(* Logix 5000 project; controller CLASE_1 Emulate 5570 rev 28.11; software revision 28.02; part 4 of 15 *)
(* tags used below, declared in another part *)
   Inp_PV : BOOL;   // Input Signal (process variable) from Sensor
   Inp_PVBad : BOOL;   // Input Comm Status or Quality 1=Bad, 0=OK
   Inp_Target : BOOL;   // Target State of Input (Disagree Status if not in Target State)
   Inp_Sim : BOOL;   // 1=Use simulated PV (Set_SimPV); 0=Use Input (Inp_PV)
   Cfg_NoSubstPV : BOOL;   // 1=Disallow selection of Substitute PV
   Cfg_Debounce : REAL;   // Minimum time Input Sts must maintain state (sec)
   MSet_SubstPV : BOOL;   // Maintenance-Entered Substitute PV
   Set_SimPV : BOOL;   // PV used in Simulation (Inp_Sim=1)
   MCmd_SubstPV : BOOL;   // Maintenance Command to use Substitute PV (override input)
   MCmd_InpPV : BOOL;   // Maintenance Command to use Input PV (normal)
   OCmd_ResetAckAll : BOOL;   // Operator Command to Reset and Acknowledge all Alarms
   SrcQ_IO : SINT;   // Source and Quality of primary I/O (enumeration)
   SrcQ : SINT;   // Source and Quality of primary Val/Sts (enumeration)
   Val_Sts : SINT;   // Device Confirmed Sts 0=PV Good, 6=PV Bad, 7=Substitute PV
   Val_Fault : SINT;   // Device Fault Status 0=none, 16=Tgt Disagree, 34=CfgErr
   Val_Notify : SINT;   // Current Alarm Level and Acknowledgement (enumeration)
   Sts : BOOL;   // Discrete Input Status (incl. Debounce, Manual Override, if used)
   Sts_PV : BOOL;   // Discrete Input Status (actual, not subject to Override)
   Sts_SubstPV : BOOL;   // 1=Using Substitute PV (Input being overridden)
   Sts_InpPV : BOOL;   // 1=Using Input PV (normal)
   Sts_PVBad : BOOL;   // Input Comm Status/ Quality (0=OK, 1=Bad)
   Sts_MaintByp : BOOL;   // 1=Device has a Maintenance Bypass function active
   Sts_AlmInh : BOOL;   // 1=One or more Alarms Shelved, Disabled or Suppressed
   Err_Alarm : BOOL;   // 1=Error in Config: Alarm Min On Time, Shelf Time, Severity
   Sts_TgtDisagreeCmp : ALIAS FOR TgtDisagreeGate.Inp;   // Input vs. Target comparicon result 1=Disagree
   Sts_TgtDisagree : ALIAS FOR TgtDisagree.Inp;   // 1=Input is not in Target state
   Rdy_SubstPV : BOOL;   // 1=Ready for MCmd_SubstPV
   Rdy_InpPV : BOOL;   // 1=Ready for MCmd_InpPV
   Rdy_ResetAckAll : BOOL;   // 1=At least one Alarm requires Acknowledgement
   P_DIn : BOOL;   // Unique Parameter Name for auto - discovery
   TgtDisagree : P_Alarm;   // Target Disagree Alarm
   Wrk_FallT : TIMER;   // Timer to ensure Status LOW time on falling edge
   Wrk_RiseT : TIMER;   // Timer to ensure Status HIGH time on rising edge
   Wrk_SubstPV : BOOL;   // Internal flag: Using Substitute PV
   Cfg_1StText : STRING_8;   // Text to display in PV=1 State
   Cfg_0StText : STRING_8;   // Text to display in PV=0 State
   Wrk_Fault : SINT;   // Buffer for building Val_Fault
   Wrk_Status : SINT;   // Buffer for building Val_Sts
   Wrk_SrcQ : SINT;   // Register for building Source / Quality enumeration
   TgtDisagreeGate : P_Gate;   // Target Disagree Condition Gate/Delay
(* P_DIn, continued *)

ROUTINE Logic   (* ladder *)
// Normal Scan - status is updated and alarms are generated
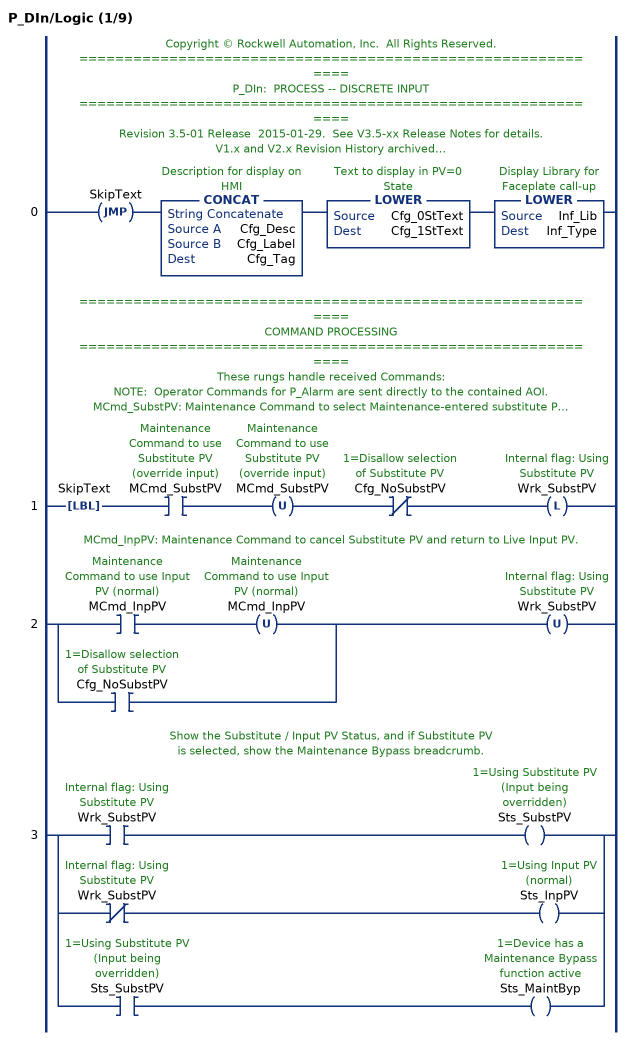
   // Copyright © Rockwell Automation, Inc.  All Rights Reserved.
   // ============================================================
   // P_DIn:  PROCESS -- DISCRETE INPUT
   // ============================================================
   // Revision 3.5-01 Release  2015-01-29.  See V3.5-xx Release Notes for details.
   // V1.x and V2.x Revision History archived.
   // V3.0-00  2013-06-30:  Added Inf_Lib. Uses P_Gate V3.0, P_Alarm V3.0.
   // V3.0-01  2013-07-30:  Modified Parameter descriptions only.
   // V3.0-02  2013-09-03:  Modified Parameter descriptions only.
   // V3.0-03  2013-10-30:  Corrected Parameter descriptions and default
   // configuration values for alarms only.
   // V3.1-00  2014-07-08:  Modified to use P_Alarm V3.1, add source/quality values (SrcQ).
   // V3.1-01  2014-09-03:  Unchanged, but using P_Alarm V3.1-01.
   // V3.1-02  2014-09-30:  Unchanged, but using P_Alarm V3.1-02.
   // V3.1-05  2016-01-22:  Unchanged, but using P_Gate V3.1-05.
   // V3.5-01  2016-01-29:  Unchanged, using P_Alarm, P_Gate V3.5-01.
   // ============================================================
   // This Instruction monitors a Discrete Input from a flow switch, motor overload,
   // or any other discrete signal, and provides:
   // *  Status, with configurable names for the 0- and 1-states
   // *  An Alarm "Gate" signal (with delay), used to enable an Alarm under appropriate process conditions
   // *  A "Target" input -- the Alarm is raised when the input is not in the same
   // state as the Target for a configurable period of time
   // * Input debounce for both the rising and falling transitions
   // * Commands to inhibit or enable alarms
   // * Monitoring of input communication status
   // * Setting of a simulated input signal for process simulation
   // * Selection of Substitute PV (by Maintenance personnel) or normal PV
   // Alarm is provided by a P_Alarm AOI instance.
   // Status gating provided by P_Gate AOI instances.
   // ============================================================
   // SHOW LOCAL STRINGS
   // ============================================================
   // The STRINGs containing the text associated with each instance of this
   // instruction cannot be Input or Output Parameters, because STRINGs are not
   //  'atomic' types. (Inputs and Outputs must be SINT, INT, DINT, REAL, or BOOL.)
   // In order to make it easier to find and configure these STRINGs, this rung
   // was added.  THE JMP (and the LBL on the following rung)
   // MUST NOT BE REMOVED!!!
   // To view the STRINGs, go to the instruction instance (in LD or FBD), RIGHT-click
   // to bring up the context menu and select "Open Instruction Logic".
   // This rung will appear with the STRING values for the selected instance.
   // You may double-click the STRING values here to modify them as well.
   // #####  V3.0-00  2013-06-30:  Added Inf_Lib.  #####
   0: JMP(SkipText)CONCAT(Cfg_Desc,Cfg_Label,Cfg_Tag)LOWER(Cfg_0StText,Cfg_1StText)LOWER(Inf_Lib,Inf_Type);
   // ============================================================
   // COMMAND PROCESSING
   // ============================================================
   // These rungs handle received Commands:
   // NOTE:  Operator Commands for P_Alarm are sent directly to the contained AOI.
   // MCmd_SubstPV: Maintenance Command to select Maintenance-entered substitute PV
   // Do not allow this Command if Cfg_NoSubstPV is set.
   1: LBL(SkipText)XIC(MCmd_SubstPV)OTU(MCmd_SubstPV)XIO(Cfg_NoSubstPV)OTL(Wrk_SubstPV);
   // MCmd_InpPV: Maintenance Command to cancel Substitute PV and return to Live Input PV.
   2: [XIC(MCmd_InpPV) OTU(MCmd_InpPV) ,XIC(Cfg_NoSubstPV) ]OTU(Wrk_SubstPV);
   // Show the Substitute / Input PV Status, and if Substitute PV
   // is selected, show the Maintenance Bypass breadcrumb.
   3: [XIC(Wrk_SubstPV) OTE(Sts_SubstPV) ,XIO(Wrk_SubstPV) OTE(Sts_InpPV) ,XIC(Sts_SubstPV) OTE(Sts_MaintByp) ];
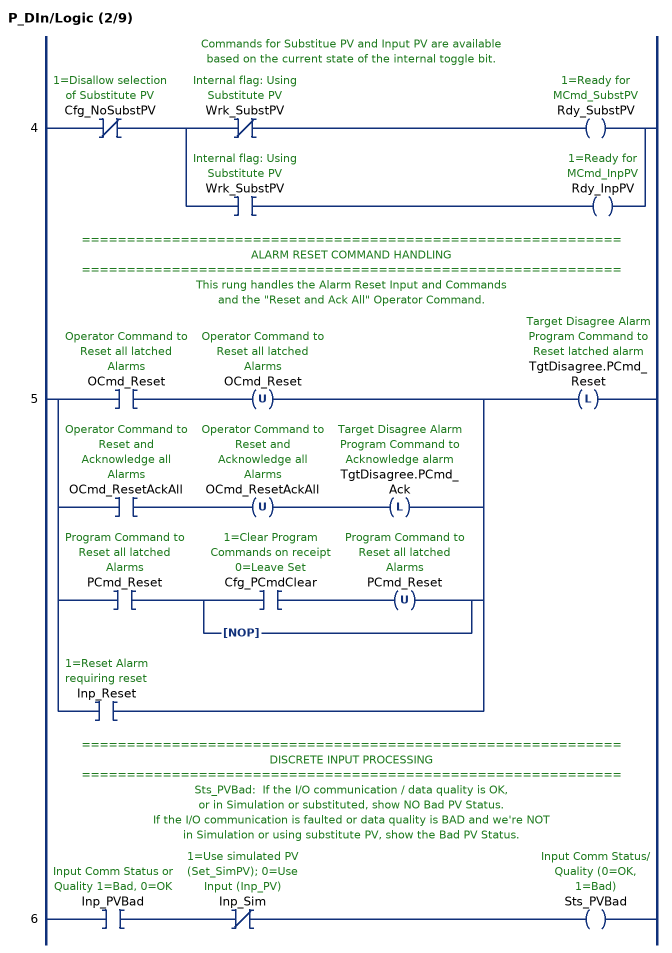
   // Commands for Substitue PV and Input PV are available
   // based on the current state of the internal toggle bit.
   4: XIO(Cfg_NoSubstPV)[XIO(Wrk_SubstPV) OTE(Rdy_SubstPV) ,XIC(Wrk_SubstPV) OTE(Rdy_InpPV) ];
   // ============================================================
   // ALARM RESET COMMAND HANDLING
   // ============================================================
   // This rung handles the Alarm Reset Input and Commands
   // and the "Reset and Ack All" Operator Command.
   5: [XIC(OCmd_Reset) OTU(OCmd_Reset) ,XIC(OCmd_ResetAckAll) OTU(OCmd_ResetAckAll) OTL(TgtDisagree.PCmd_Ack) ,XIC(PCmd_Reset) [XIC(Cfg_PCmdClear) OTU(PCmd_Reset) ,NOP() ] ,XIC(Inp_Reset) ]OTL(TgtDisagree.PCmd_Reset);
   // ============================================================
   // DISCRETE INPUT PROCESSING
   // ============================================================
   // Sts_PVBad:  If the I/O communication / data quality is OK,
   // or in Simulation or substituted, show NO Bad PV Status.
   // If the I/O communication is faulted or data quality is BAD and we're NOT
   // in Simulation or using substitute PV, show the Bad PV Status.
   6: XIC(Inp_PVBad)XIO(Inp_Sim)OTE(Sts_PVBad);
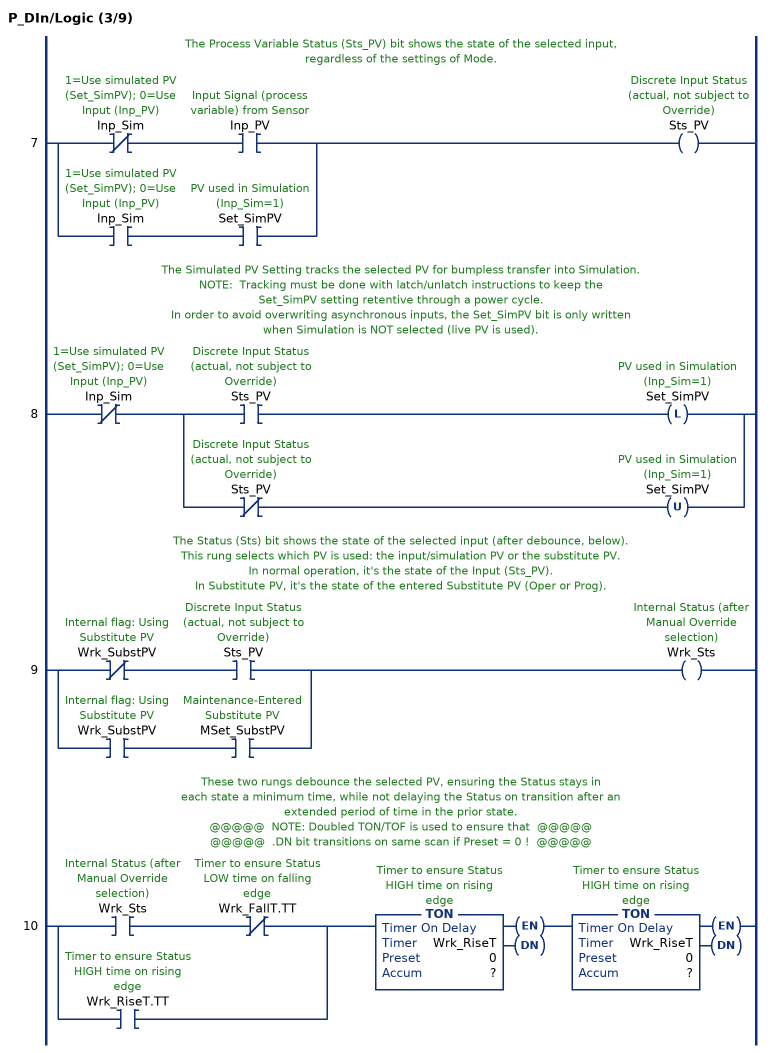
   // The Process Variable Status (Sts_PV) bit shows the state of the selected input,
   // regardless of the settings of Mode.
   7: [XIO(Inp_Sim) XIC(Inp_PV) ,XIC(Inp_Sim) XIC(Set_SimPV) ]OTE(Sts_PV);
   // The Simulated PV Setting tracks the selected PV for bumpless transfer into Simulation.
   // NOTE:  Tracking must be done with latch/unlatch instructions to keep the
   // Set_SimPV setting retentive through a power cycle.
   // In order to avoid overwriting asynchronous inputs, the Set_SimPV bit is only written
   // when Simulation is NOT selected (live PV is used).
   8: XIO(Inp_Sim)[XIC(Sts_PV) OTL(Set_SimPV) ,XIO(Sts_PV) OTU(Set_SimPV) ];
   // The Status (Sts) bit shows the state of the selected input (after debounce, below).
   // This rung selects which PV is used: the input/simulation PV or the substitute PV.
   // In normal operation, it's the state of the Input (Sts_PV).
   // In Substitute PV, it's the state of the entered Substitute PV (Oper or Prog).
   9: [XIO(Wrk_SubstPV) XIC(Sts_PV) ,XIC(Wrk_SubstPV) XIC(MSet_SubstPV) ]OTE(Wrk_Sts);
   // These two rungs debounce the selected PV, ensuring the Status stays in
   // each state a minimum time, while not delaying the Status on transition after an
   // extended period of time in the prior state.
   // @@@@@  NOTE: Doubled TON/TOF is used to ensure that  @@@@@
   // @@@@@  .DN bit transitions on same scan if Preset = 0 !  @@@@@
   10: [XIC(Wrk_Sts) XIO(Wrk_FallT.TT) ,XIC(Wrk_RiseT.TT) ]TON(Wrk_RiseT,?,?)TON(Wrk_RiseT,?,?);
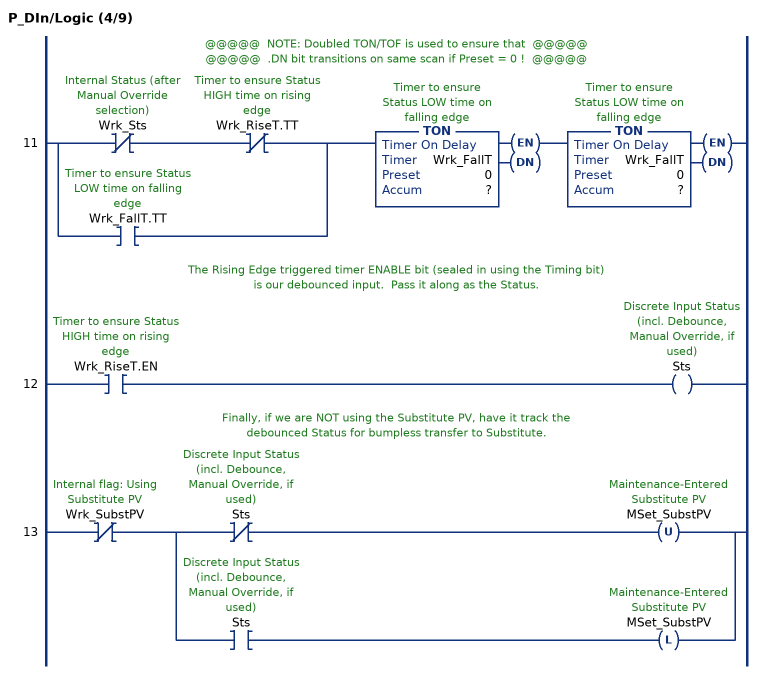
   // @@@@@  NOTE: Doubled TON/TOF is used to ensure that  @@@@@
   // @@@@@  .DN bit transitions on same scan if Preset = 0 !  @@@@@
   11: [XIO(Wrk_Sts) XIO(Wrk_RiseT.TT) ,XIC(Wrk_FallT.TT) ]TON(Wrk_FallT,?,?)TON(Wrk_FallT,?,?);
   // The Rising Edge triggered timer ENABLE bit (sealed in using the Timing bit)
   // is our debounced input.  Pass it along as the Status.
   12: XIC(Wrk_RiseT.EN)OTE(Sts);
   // Finally, if we are NOT using the Substitute PV, have it track the
   // debounced Status for bumpless transfer to Substitute.
   13: XIO(Wrk_SubstPV)[XIO(Sts) OTU(MSet_SubstPV) ,XIC(Sts) OTL(MSet_SubstPV) ];
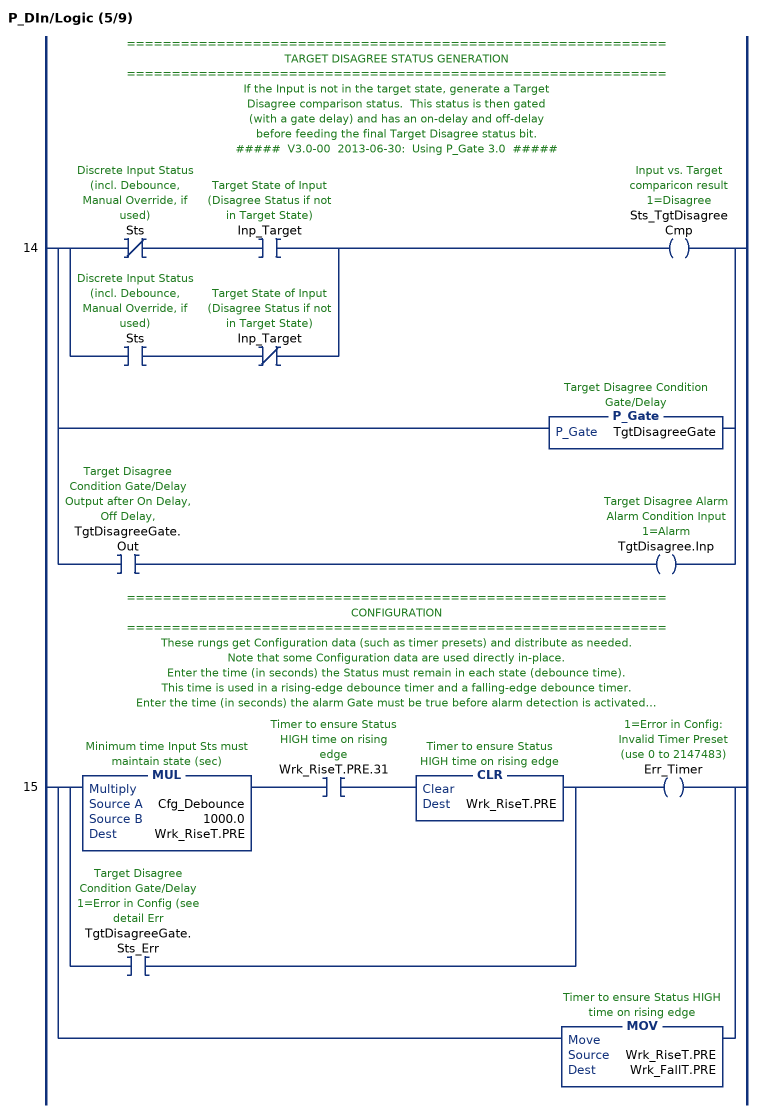
   // ============================================================
   // TARGET DISAGREE STATUS GENERATION
   // ============================================================
   // If the Input is not in the target state, generate a Target
   // Disagree comparison status.  This status is then gated
   // (with a gate delay) and has an on-delay and off-delay
   // before feeding the final Target Disagree status bit.
   // #####  V3.0-00  2013-06-30:  Using P_Gate 3.0  #####
   14: [[XIO(Sts) XIC(Inp_Target) ,XIC(Sts) XIO(Inp_Target) ] OTE(Sts_TgtDisagreeCmp) ,P_Gate(TgtDisagreeGate) ,XIC(TgtDisagreeGate.Out) OTE(TgtDisagree.Inp) ];
   // ============================================================
   // CONFIGURATION
   // ============================================================
   // These rungs get Configuration data (such as timer presets) and distribute as needed.
   // Note that some Configuration data are used directly in-place.
   // Enter the time (in seconds) the Status must remain in each state (debounce time).
   // This time is used in a rising-edge debounce timer and a falling-edge debounce timer.
   // Enter the time (in seconds) the alarm Gate must be true before alarm detection is activated.
   // Enter the On-Delay and Off-Delay times (in seconds) for the Target Disagree Status
   // (which feeds the Target Disagree Alarm).
   // If the timer preset calcuated wraps negative (more than 2.14... million seconds), then establish
   // a valid limit value for the Preset.  Note that a negative timer preset will fault the controller!!!
   // #####  V3.0-00  2013-06-30:  Using P_Gate 3.0  #####
   15: [[MUL(Cfg_Debounce,1000.0,Wrk_RiseT.PRE) XIC(Wrk_RiseT.PRE.31) CLR(Wrk_RiseT.PRE) ,XIC(TgtDisagreeGate.Sts_Err) ] OTE(Err_Timer) ,MOV(Wrk_RiseT.PRE,Wrk_FallT.PRE) ];
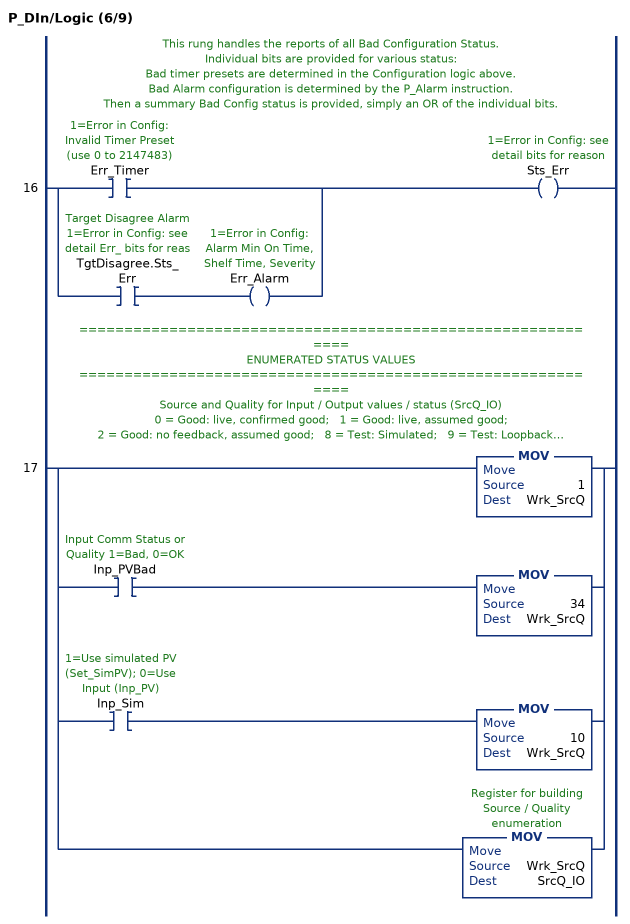
   // This rung handles the reports of all Bad Configuration Status.
   // Individual bits are provided for various status:
   // Bad timer presets are determined in the Configuration logic above.
   // Bad Alarm configuration is determined by the P_Alarm instruction.
   // Then a summary Bad Config status is provided, simply an OR of the individual bits.
   16: [XIC(Err_Timer) ,XIC(TgtDisagree.Sts_Err) OTE(Err_Alarm) ]OTE(Sts_Err);
   // ============================================================
   // ENUMERATED STATUS VALUES
   // ============================================================
   // Source and Quality for Input / Output values / status (SrcQ_IO)
   // 0 = Good: live, confirmed good;   1 = Good: live, assumed good;
   // 2 = Good: no feedback, assumed good;   8 = Test: Simulated;   9 = Test: Loopback;
   // 10 = Test: Manually Entered;   16 = Uncertain: Live, off-spec;
   // 17 = Uncertain, Substituted at Device / Bus;   18 = Uncertain, Substituted at AOI;
   // 19 = Uncertain, using last known good;    20 = Uncertain, using replacement value;
   // 32 = Bad, Signal Failure;   33 = Bad, Channel Fault;
   // 34 = Bad, Module / Comms Fault;   35 = Bad, Invalid Configuration
   // #####  V3.1-00  2014-06-30:  Added rung for Source/Quality enumerations.  #####
   17: [MOV(1,Wrk_SrcQ) ,XIC(Inp_PVBad) MOV(34,Wrk_SrcQ) ,XIC(Inp_Sim) MOV(10,Wrk_SrcQ) ,MOV(Wrk_SrcQ,SrcQ_IO) ];
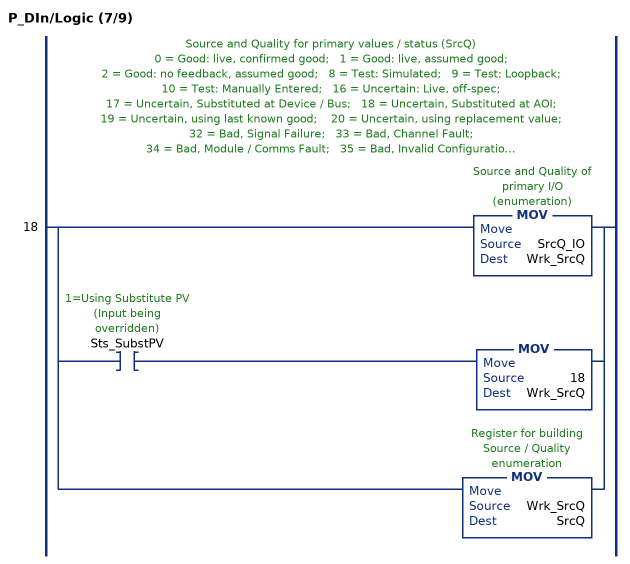
   // Source and Quality for primary values / status (SrcQ)
   // 0 = Good: live, confirmed good;   1 = Good: live, assumed good;
   // 2 = Good: no feedback, assumed good;   8 = Test: Simulated;   9 = Test: Loopback;
   // 10 = Test: Manually Entered;   16 = Uncertain: Live, off-spec;
   // 17 = Uncertain, Substituted at Device / Bus;   18 = Uncertain, Substituted at AOI;
   // 19 = Uncertain, using last known good;    20 = Uncertain, using replacement value;
   // 32 = Bad, Signal Failure;   33 = Bad, Channel Fault;
   // 34 = Bad, Module / Comms Fault;   35 = Bad, Invalid Configuration
   // #####  V3.1-00  2014-06-30:  Added rung for Source/Quality enumerations.  #####
   18: [MOV(SrcQ_IO,Wrk_SrcQ) ,XIC(Sts_SubstPV) MOV(18,Wrk_SrcQ) ,MOV(Wrk_SrcQ,SrcQ) ];
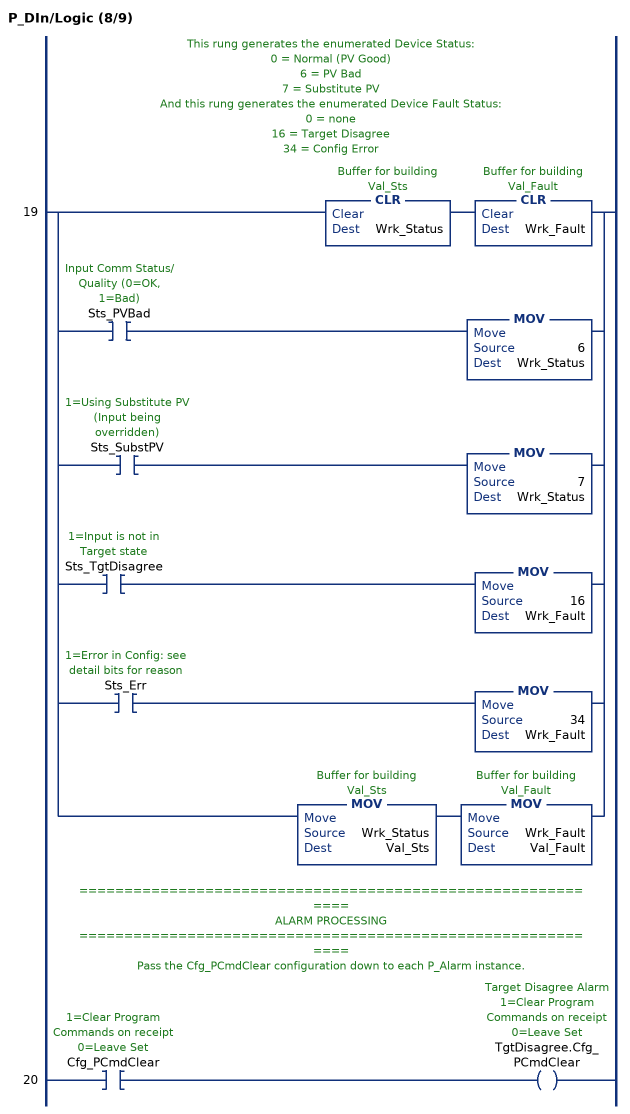
   // This rung generates the enumerated Device Status:
   // 0 = Normal (PV Good)
   // 6 = PV Bad
   // 7 = Substitute PV
   // And this rung generates the enumerated Device Fault Status:
   // 0 = none
   // 16 = Target Disagree
   // 34 = Config Error
   19: [CLR(Wrk_Status) CLR(Wrk_Fault) ,XIC(Sts_PVBad) MOV(6,Wrk_Status) ,XIC(Sts_SubstPV) MOV(7,Wrk_Status) ,XIC(Sts_TgtDisagree) MOV(16,Wrk_Fault) ,XIC(Sts_Err) MOV(34,Wrk_Fault) ,MOV(Wrk_Status,Val_Sts) MOV(Wrk_Fault,Val_Fault) ];
   // ============================================================
   // ALARM PROCESSING
   // ============================================================
   // Pass the Cfg_PCmdClear configuration down to each P_Alarm instance.
   20: XIC(Cfg_PCmdClear)OTE(TgtDisagree.Cfg_PCmdClear);
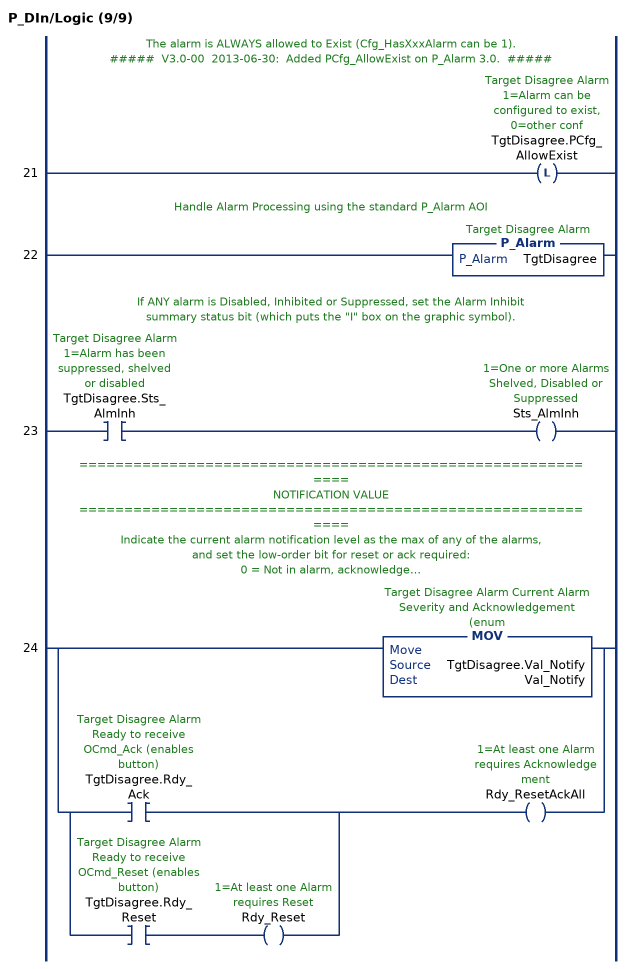
   // The alarm is ALWAYS allowed to Exist (Cfg_HasXxxAlarm can be 1).
   // #####  V3.0-00  2013-06-30:  Added PCfg_AllowExist on P_Alarm 3.0.  #####
   21: OTL(TgtDisagree.PCfg_AllowExist);
   // Handle Alarm Processing using the standard P_Alarm AOI
   22: P_Alarm(TgtDisagree);
   // If ANY alarm is Disabled, Inhibited or Suppressed, set the Alarm Inhibit
   // summary status bit (which puts the "I" box on the graphic symbol).
   23: XIC(TgtDisagree.Sts_AlmInh)OTE(Sts_AlmInh);
   // ============================================================
   // NOTIFICATION VALUE
   // ============================================================
   // Indicate the current alarm notification level as the max of any of the alarms,
   // and set the low-order bit for reset or ack required:
   // 0 = Not in alarm, acknowledged
   // 1 = Not in alarm, unacknowledged or reset required
   // 2 = Low severity alarm, acknowledged
   // 3 = Low severity alarm, unacknowledged
   // 4 = Medium severity alarm, acknowledged
   // 5 = Medium severity alarm, unacknowledged
   // 6 = High severity alarm, acknowledged
   // 7 = High severity alarm, unacknowledged
   // 8 = Urgent severity alarm, acknowledged
   // 9 = Urgent severity alarm, unacknowledged
   // #####  V3.1-00  2014-06-30:  Separated Reset Reqd functions from Val_Notify  #####
   24: [MOV(TgtDisagree.Val_Notify,Val_Notify) ,[XIC(TgtDisagree.Rdy_Ack) ,XIC(TgtDisagree.Rdy_Reset) OTE(Rdy_Reset) ] OTE(Rdy_ResetAckAll) ];
END_ROUTINE

ROUTINE Prescan   (* ladder *)
// Clear "lurking" Commands
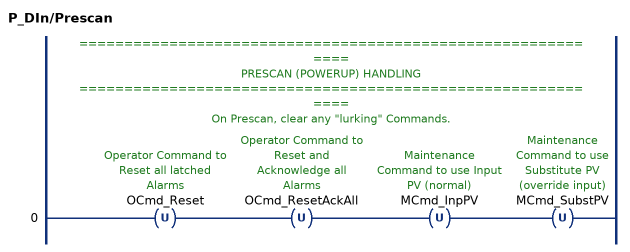
   // ============================================================
   // PRESCAN (POWERUP) HANDLING
   // ============================================================
   // On Prescan, clear any "lurking" Commands.
   0: OTU(OCmd_Reset)OTU(OCmd_ResetAckAll)OTU(MCmd_InpPV)OTU(MCmd_SubstPV);
END_ROUTINE
END_ADD_ON_INSTRUCTION

ADD_ON_INSTRUCTION P_FT_Primer_Orden_AOI   (* revision 1.0 *)
// Simula el comportamiento de una Función de Transferencia de primer orden.
// G(s) = Kp/(Tao*s + 1)
VAR_INPUT
   Kp : REAL; {visible}   // Ganancia proporcional de la FT.
   Tao : REAL; {visible}   // Tao de la FT (en segundos).
   Inp_Sistema : REAL; {visible}   // Entrada de la FT.
END_VAR
VAR_OUTPUT
   Out_Sistema : REAL; {visible}   // Salida de la FT.
END_VAR
VAR_INPUT
   Tiempo_muerto : REAL; {visible}   // Tiempo muerto (en segundos).
   Inp_Disturbio : REAL; {visible}   // Permite simular un disturbio en el sistema.
   FT_EnableIN : BOOL := 1; {visible}   // Bit para ejecutar algoritmo de la FT.
   FT_Bias : REAL; {visible}   // Simula condición de proceso. (In*Gain) + Bias.
END_VAR
VAR
   DEDT_01 : DEADTIME := (Gain := 1.0, RTSTime := 1); {access None}
   LDLG_01 : LEAD_LAG := (Gain := 1.0, RTSTime := 1); {access None}
   FT : LEAD_LAG := (Gain := 1.0, RTSTime := 1);   // Simula FT de Primer Orden.
   Tm : DEADTIME := (Gain := 1.0, RTSTime := 1); {access None}   // Simula Tiempo muerto.
   Tm_muestreo : REAL[1000]; {access None}   // Array para guardar valores previos al Tiempo muestro.
   ADD_01 : FBD_MATH; {access None}
   __l01D9873C3019917B : REAL; {access None}
   __l01D9933530198D26 : BOOL; {access None}
   __l01D9DEFB3019BCF5 : REAL; {access None}
   __l01D9CACD3019D0A3 : REAL; {access None}
   __l01D9EFCA30199939 : REAL; {access None}
   __l01D9E71B3019C2AC : REAL; {access None}
   __l01D9EBF23019A41E : REAL; {access None}
END_VAR

ROUTINE Logic   (* function block diagram *)
   SHEET 1
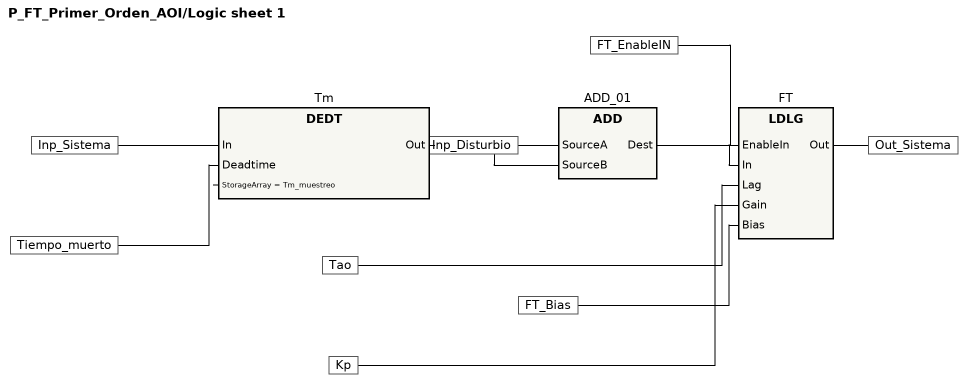
   Tm : DEDT(In := Inp_Sistema, Deadtime := Tiempo_muerto, StorageArray := Tm_muestreo);
   ADD_01 : ADD(SourceA := Inp_Disturbio, SourceB := Tm.Out);
   FT : LDLG(EnableIn := FT_EnableIN, In := ADD_01.Dest, Lag := Tao, Gain := Kp, Bias := FT_Bias);
   Out_Sistema := FT.Out;
END_ROUTINE
END_ADD_ON_INSTRUCTION

ADD_ON_INSTRUCTION P_Gate   (* revision 3.5 01 Release, vendor Rockwell Automation, ExecutePrescan, ExecuteEnableInFalse *)
// Condition Gate/Delay
// Revision note:
// See V3.5-xx Release Notes for details. Unchanged, up-rev only for V3.5 Library.
// Help:
// Copyright © Rockwell Automation, Inc.  All Rights Reserved.
// This Instruction provides a "gate" for a discrete Input signal and
// provides on-delay and off-delay timing for the gated signal.
// When the Gate input is true, the instruction Input is passed through
// to the Output, with on-delay and off-delay timing applied.
// When the Gate input is false, the Output is kept off
// (note: off-delay still applies!)
// This instruction is usually used between a comparison
// (analog threshold with deadband or discrete logic)
// and a P_Alarm instance, but may be used as a
// gated on-delay/off-delay timer generally.
// When EnableIn  is FALSE (e.g., on a false LD rung),
// the Input "Inp" is inverted.  Note that the Gate
// input (Inp_Gate) is NOT inverted!!!
VAR_INPUT
   Inp : BOOL; {visible}   // Input Condition: e.g., result of comparison
   Inp_Gate : BOOL := 1; {visible}   // Gate Input: 1=enable On Delay / Off Delay after Gate Delay, 0=disable
   Cfg_GateDly : DINT;   // Gate Delay (s): time after Gate Input true to enable On/Off Delay
   Cfg_OnDly : DINT;   // On Delay (s): If Gate Delay done, time Inp must be true to set Out true
   Cfg_OffDly : DINT;   // Off Delay (s): Time after Inp or Gate goes to 0 for Out to go to 0
END_VAR
VAR_OUTPUT
   Out : BOOL; {access Read Only, visible}   // Output after On Delay, Off Delay, enabled by Gate
   Sts_Gate : BOOL; {access Read Only, visible}   // 1=Gate Delay done, Output is enabled
   Sts_Err : BOOL; {access Read Only, visible}   // 1=Error in Config (see detail Err_ bits for reason), display icon
   Err_Timer : BOOL; {access Read Only}   // 1=Error in Config: On Delay, Off Delay, Gate Delay Time Invalid (use 0 to 2147483 s)
   P_Gate : BOOL;   // Unique Parameter Name for auto - discovery
END_VAR
VAR
   Wrk_OffDlyT : TIMER; {access Read Only}   // Off Delay Timer
   Wrk_OnDlyT : TIMER; {access Read Only}   // On Delay Timer
   Wrk_GateT : TIMER; {access Read Only}   // Gate Delay Timer
   Cfg_InpCond : STRING_20 := 'Input Condition';   // Displayed text of P_Gate's Input (Inp) Condition
   Inf_Lib : STRING_12 := 'RA-BAS'; {access Read Only}   // Display Library for Faceplate call-up
   Inf_Type : STRING_16 := 'P_Gate'; {access Read Only}   // Must contain AOI name, used for HMI and Information S/W
   Cfg_GateCond : STRING_20 := 'Gating Condition';   // Displayed text of P_Gate's Gating (Inp_Gate) Condition
   Inf_Tab : SINT;   // Tab to display (FTView ME)
END_VAR

ROUTINE EnableInFalse   (* ladder *)
// Same as main Logic routine, except Inp is inverted (for use in LD logic)  (Inp_Gate is NOT inverted!!!)
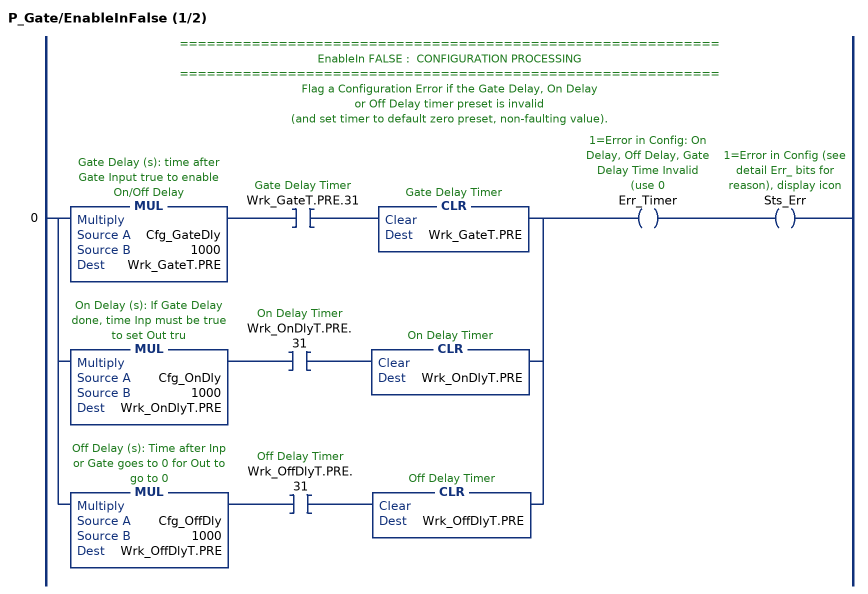
   // ============================================================
   // EnableIn FALSE :  CONFIGURATION PROCESSING
   // ============================================================
   // Flag a Configuration Error if the Gate Delay, On Delay
   // or Off Delay timer preset is invalid
   // (and set timer to default zero preset, non-faulting value).
   0: [MUL(Cfg_GateDly,1000,Wrk_GateT.PRE) XIC(Wrk_GateT.PRE.31) CLR(Wrk_GateT.PRE) ,MUL(Cfg_OnDly,1000,Wrk_OnDlyT.PRE) XIC(Wrk_OnDlyT.PRE.31) CLR(Wrk_OnDlyT.PRE) ,MUL(Cfg_OffDly,1000,Wrk_OffDlyT.PRE) XIC(Wrk_OffDlyT.PRE.31) CLR(Wrk_OffDlyT.PRE) ]OTE(Err_Timer)OTE(Sts_Err);
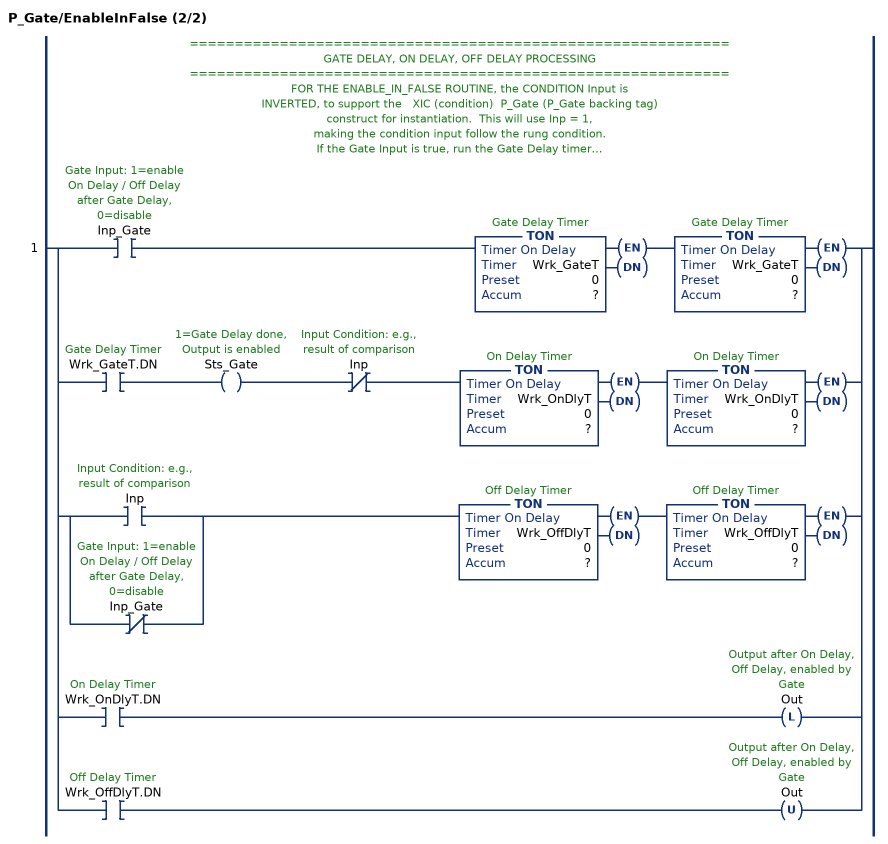
   // ============================================================
   // GATE DELAY, ON DELAY, OFF DELAY PROCESSING
   // ============================================================
   // FOR THE ENABLE_IN_FALSE ROUTINE, the CONDITION Input is
   // INVERTED, to support the   XIC (condition)  P_Gate (P_Gate backing tag)
   // construct for instantiation.  This will use Inp = 1,
   // making the condition input follow the rung condition.
   // If the Gate Input is true, run the Gate Delay timer.
   // Once the Gate Delay is complete, enable the
   // On Delay and Off Delay that follow the INVERTED input.
   // Report the Gate Delay status and the final Output status (after all delays).
   // @@@@@  NOTE: Doubled TONs are used to ensure that  @@@@@
   // @@@@@  .DN bit transitions on same scan if Preset = 0 !  @@@@@
   1: [XIC(Inp_Gate) TON(Wrk_GateT,?,?) TON(Wrk_GateT,?,?) ,XIC(Wrk_GateT.DN) OTE(Sts_Gate) XIO(Inp) TON(Wrk_OnDlyT,?,?) TON(Wrk_OnDlyT,?,?) ,[XIC(Inp) ,XIO(Inp_Gate) ] TON(Wrk_OffDlyT,?,?) TON(Wrk_OffDlyT,?,?) ,XIC(Wrk_OnDlyT.DN) OTL(Out) ,XIC(Wrk_OffDlyT.DN) OTU(Out) ];
END_ROUTINE

ROUTINE Logic   (* ladder *)
// Gate the input and apply on-delay and off-delay timing
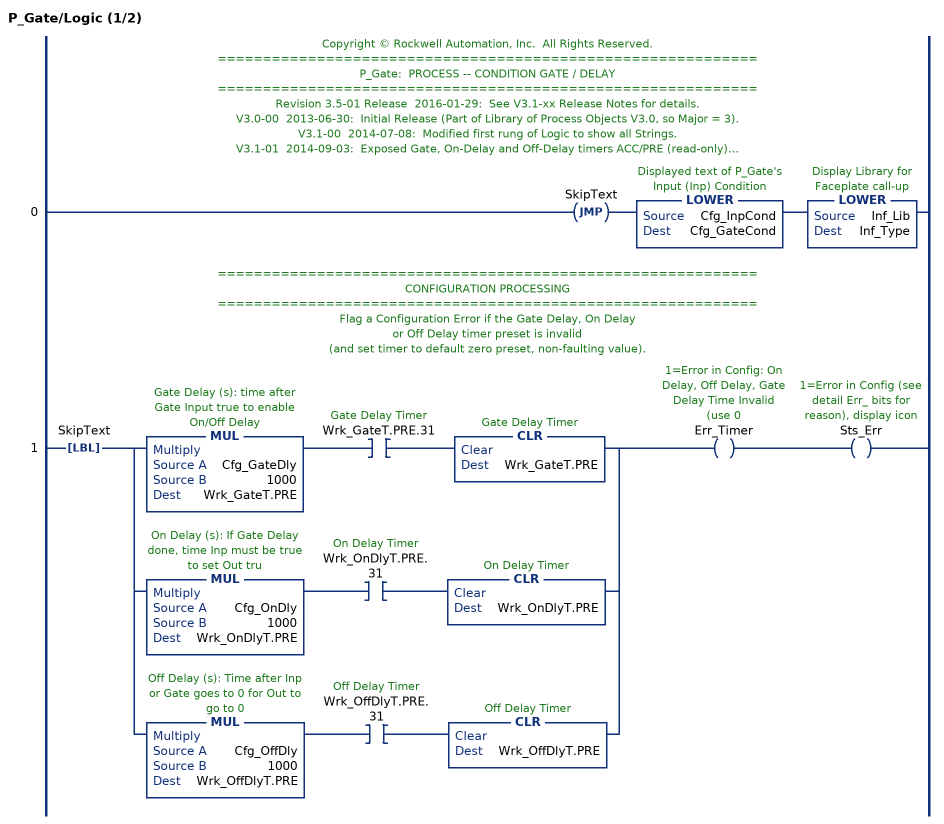
   // Copyright © Rockwell Automation, Inc.  All Rights Reserved.
   // ============================================================
   // P_Gate:  PROCESS -- CONDITION GATE / DELAY
   // ============================================================
   // Revision 3.5-01 Release  2016-01-29:  See V3.1-xx Release Notes for details.
   // V3.0-00  2013-06-30:  Initial Release (Part of Library of Process Objects V3.0, so Major = 3).
   // V3.1-00  2014-07-08:  Modified first rung of Logic to show all Strings.
   // V3.1-01  2014-09-03:  Exposed Gate, On-Delay and Off-Delay timers ACC/PRE (read-only).
   // V3.1-05  2016-01-22:  Corrected logic when using analog threshold with deadband.
   // V3.5-01  2016-01-29:  Unchanged, up-rev only for V3.5 Library.
   // ============================================================
   // This Instruction provides a "gate" for a discrete Input signal and
   // provides on-delay and off-delay timing for the gated signal.
   // When the Gate input is true, the instruction Input is passed through
   // to the Output, with on-delay and off-delay timing applied.
   // When the Gate input is false, the Output is kept off
   // (note: off-delay still applies!)
   // This instruction is usually used between a comparison
   // (analog threshold with deadband or discrete logic)
   // and a P_Alarm instance, but may be used as a
   // gated on-delay/off-delay timer generally.
   // When EnableIn  is FALSE (e.g., on a false LD rung),
   // the Input "Inp" is inverted.  Note that the Gate
   // input (Inp_Gate) is NOT inverted!!!
   // ============================================================
   // SHOW LOCAL STRINGS
   // ============================================================
   // The STRINGs containing the text associated with each instance of this
   // instruction cannot be Input or Output Parameters, because STRINGs are not
   //  'atomic' types. (Inputs and Outputs must be SINT, INT, DINT, REAL, or BOOL.)
   // In order to make it easier to find and configure these STRINGs, this rung
   // was added.  THE JMP (and the LBL on the following rung)
   // MUST NOT BE REMOVED!!!
   // To view the STRINGs, go to the instruction instance (in LD or FBD), RIGHT-click
   // to bring up the context menu and select "Open Instruction Logic".
   // This rung will appear with the STRING values for the selected instance.
   // You may double-click the STRING values here to modify them as well.
   // #####  V3.1-00  2014-07-08: Added Inf_Type to displayed Strings  #####
   0: JMP(SkipText)LOWER(Cfg_InpCond,Cfg_GateCond)LOWER(Inf_Lib,Inf_Type);
   // ============================================================
   // CONFIGURATION PROCESSING
   // ============================================================
   // Flag a Configuration Error if the Gate Delay, On Delay
   // or Off Delay timer preset is invalid
   // (and set timer to default zero preset, non-faulting value).
   1: LBL(SkipText)[MUL(Cfg_GateDly,1000,Wrk_GateT.PRE) XIC(Wrk_GateT.PRE.31) CLR(Wrk_GateT.PRE) ,MUL(Cfg_OnDly,1000,Wrk_OnDlyT.PRE) XIC(Wrk_OnDlyT.PRE.31) CLR(Wrk_OnDlyT.PRE) ,MUL(Cfg_OffDly,1000,Wrk_OffDlyT.PRE) XIC(Wrk_OffDlyT.PRE.31) CLR(Wrk_OffDlyT.PRE) ]OTE(Err_Timer)OTE(Sts_Err);
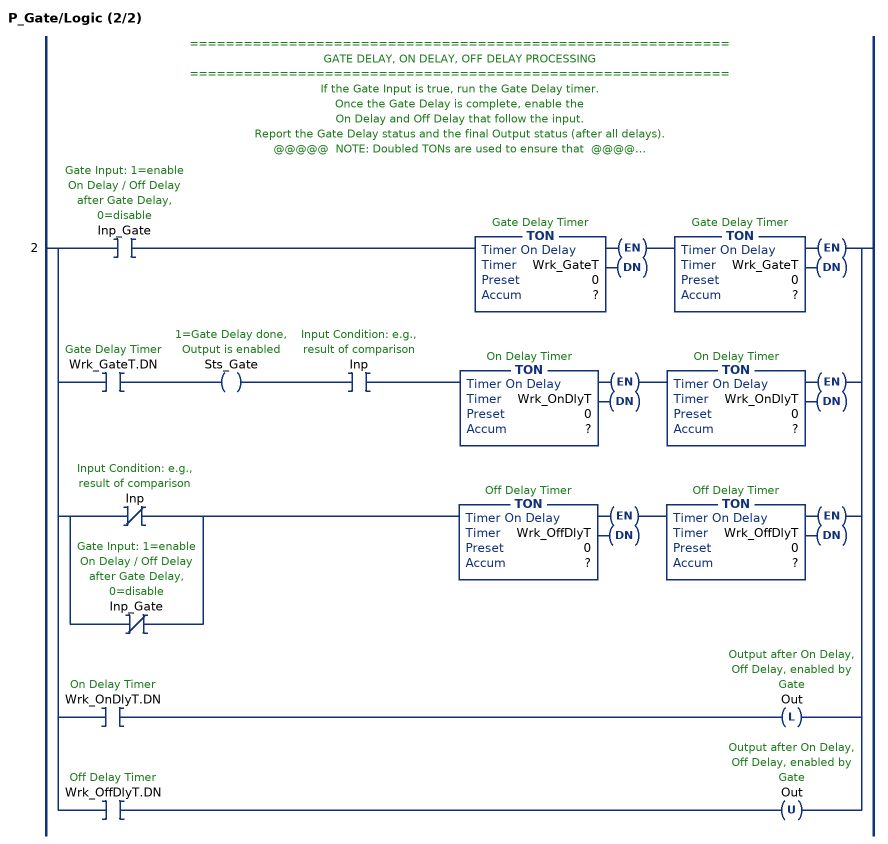
   // ============================================================
   // GATE DELAY, ON DELAY, OFF DELAY PROCESSING
   // ============================================================
   // If the Gate Input is true, run the Gate Delay timer.
   // Once the Gate Delay is complete, enable the
   // On Delay and Off Delay that follow the input.
   // Report the Gate Delay status and the final Output status (after all delays).
   // @@@@@  NOTE: Doubled TONs are used to ensure that  @@@@@
   // @@@@@  .DN bit transitions on same scan if Preset = 0 !  @@@@@
   2: [XIC(Inp_Gate) TON(Wrk_GateT,?,?) TON(Wrk_GateT,?,?) ,XIC(Wrk_GateT.DN) OTE(Sts_Gate) XIC(Inp) TON(Wrk_OnDlyT,?,?) TON(Wrk_OnDlyT,?,?) ,[XIO(Inp) ,XIO(Inp_Gate) ] TON(Wrk_OffDlyT,?,?) TON(Wrk_OffDlyT,?,?) ,XIC(Wrk_OnDlyT.DN) OTL(Out) ,XIC(Wrk_OffDlyT.DN) OTU(Out) ];
END_ROUTINE

ROUTINE Prescan   (* ladder *)
// Set the Gate Input to 1 (default value) on prescan
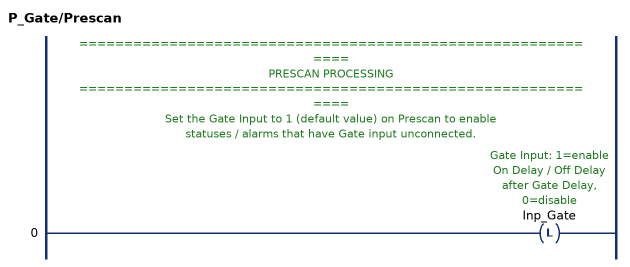
   // ============================================================
   // PRESCAN PROCESSING
   // ============================================================
   // Set the Gate Input to 1 (default value) on Prescan to enable
   // statuses / alarms that have Gate input unconnected.
   0: OTL(Inp_Gate);
END_ROUTINE
END_ADD_ON_INSTRUCTION

ADD_ON_INSTRUCTION P_Intlk   (* revision 3.5 05 Release, vendor Rockwell Automation, ExecutePrescan, ExecuteEnableInFalse *)
// Interlocks
// Revision note:
// See V3.5-xx Release Notes for details. Changed Nav Tags to user-defined STRING_NavTag type. Modified to maintain First Out indication until next stop.
// Help:
// Copyright © Rockwell Automation, Inc.  All Rights Reserved.
// This Instruction monitors up to 16 Interlock conditions.  It provides these features:
// *  The "OK" state of each Interlock Input is configurable.  By default,
//     each Input is 1 to trip, 0 when OK to run.
// *  Interlocks may be configured as Latched.  Latched Interlocks
//     require a Reset Command to clear.  The latching function can be
//     inhibited via a Latch Defeat input, for example, to avoid latching
//     Interlocks for a stopped motor.
// *  Interlocks may be configured as Bypassable; Non-Bypassable
//     Interlocks are reported separately so the destination object can
//     decide whether to bypass (ignore) bypassable interlocks, such
//     as in Maintenance Mode.
// *  First-Out reporting indicates the first condition that caused the
//     running equipment to be tripped.
// *  For each Interlock condition, a Tag may be defined for navigation.
//     Clicking the Interlock description will call up the associated Tag's
//     Faceplate.
VAR_INPUT
   Inp_Intlk00 : ALIAS FOR Wrk_Inp.0; {visible}   // Interlock Cond. 00, Stop if not in configured OK state
   Inp_Intlk01 : ALIAS FOR Wrk_Inp.1; {visible}   // Interlock Cond. 01, Stop if not in configured OK state
   Inp_Intlk02 : ALIAS FOR Wrk_Inp.2; {visible}   // Interlock Cond. 02, Stop if not in configured OK state
   Inp_Intlk03 : ALIAS FOR Wrk_Inp.3; {visible}   // Interlock Cond. 03, Stop if not in configured OK state
   Inp_Intlk04 : ALIAS FOR Wrk_Inp.4; {visible}   // Interlock Cond. 04, Stop if not in configured OK state
   Inp_Intlk05 : ALIAS FOR Wrk_Inp.5; {visible}   // Interlock Cond. 05, Stop if not in configured OK state
   Inp_Intlk06 : ALIAS FOR Wrk_Inp.6; {visible}   // Interlock Cond. 06, Stop if not in configured OK state
   Inp_Intlk07 : ALIAS FOR Wrk_Inp.7; {visible}   // Interlock Cond. 07, Stop if not in configured OK state
   Inp_Intlk08 : ALIAS FOR Wrk_Inp.8;   // Interlock Cond. 08, Stop if not in configured OK state
   Inp_Intlk09 : ALIAS FOR Wrk_Inp.9;   // Interlock Cond. 09, Stop if not in configured OK state
   Inp_Intlk10 : ALIAS FOR Wrk_Inp.10;   // Interlock Cond. 10, Stop if not in configured OK state
   Inp_Intlk11 : ALIAS FOR Wrk_Inp.11;   // Interlock Cond. 11, Stop if not in configured OK state
   Inp_Intlk12 : ALIAS FOR Wrk_Inp.12;   // Interlock Cond. 12, Stop if not in configured OK state
   Inp_Intlk13 : ALIAS FOR Wrk_Inp.13;   // Interlock Cond. 13, Stop if not in configured OK state
   Inp_Intlk14 : ALIAS FOR Wrk_Inp.14;   // Interlock Cond. 14, Stop if not in configured OK state
   Inp_Intlk15 : ALIAS FOR Wrk_Inp.15;   // Interlock Cond. 15, Stop if not in configured OK state
   Inp_BypActive : BOOL; {visible}   // 1=Interlock Bypassing is currently active
   Inp_LatchDefeat : BOOL; {visible}   // Latch Defeat 1=Do not latch inputs even if configured for latching
   Inp_Reset : BOOL; {visible}   // 1=Reset Latched Interlocks and First-Out
   Cfg_OKState : INT;   // Bits indicate which state (0 or 1) of each input is OK to run
   Cfg_Latched : INT;   // Set bits indicate which conditions are latched (sealed in)
   Cfg_Bypassable : INT;   // Set bits indicate which conditions can be bypassed
   Cfg_HasNav : INT;   // Set bits indicate which Navigation buttons are enabled
   Cfg_PCmdClear : BOOL := 1;   // 1=Clear Program Commands on receipt 0=Leave Set
   MSet_Bypass00 : ALIAS FOR Wrk_MSet.0;   // Maint. Bypass Toggle for Interlock Cond. 00: 1=Bypass
   MSet_Bypass01 : ALIAS FOR Wrk_MSet.1;   // Maint. Bypass Toggle for Interlock Cond. 0`: 1=Bypass
   MSet_Bypass02 : ALIAS FOR Wrk_MSet.2;   // Maint. Bypass Toggle for Interlock Cond. 02: 1=Bypass
   MSet_Bypass03 : ALIAS FOR Wrk_MSet.3;   // Maint. Bypass Toggle for Interlock Cond. 03: 1=Bypass
   MSet_Bypass04 : ALIAS FOR Wrk_MSet.4;   // Maint. Bypass Toggle for Interlock Cond. 04: 1=Bypass
   MSet_Bypass05 : ALIAS FOR Wrk_MSet.5;   // Maint. Bypass Toggle for Interlock Cond. 05: 1=Bypass
   MSet_Bypass06 : ALIAS FOR Wrk_MSet.6;   // Maint. Bypass Toggle for Interlock Cond. 06: 1=Bypass
   MSet_Bypass07 : ALIAS FOR Wrk_MSet.7;   // Maint. Bypass Toggle for Interlock Cond. 07: 1=Bypass
   MSet_Bypass08 : ALIAS FOR Wrk_MSet.8;   // Maint. Bypass Toggle for Interlock Cond. 08: 1=Bypass
   MSet_Bypass09 : ALIAS FOR Wrk_MSet.9;   // Maint. Bypass Toggle for Interlock Cond. 09: 1=Bypass
   MSet_Bypass10 : ALIAS FOR Wrk_MSet.10;   // Maint. Bypass Toggle for Interlock Cond. 10: 1=Bypass
   MSet_Bypass11 : ALIAS FOR Wrk_MSet.11;   // Maint. Bypass Toggle for Interlock Cond. 11: 1=Bypass
   MSet_Bypass12 : ALIAS FOR Wrk_MSet.12;   // Maint. Bypass Toggle for Interlock Cond. 12: 1=Bypass
   MSet_Bypass13 : ALIAS FOR Wrk_MSet.13;   // Maint. Bypass Toggle for Interlock Cond. 13: 1=Bypass
   MSet_Bypass14 : ALIAS FOR Wrk_MSet.14;   // Maint. Bypass Toggle for Interlock Cond. 14: 1=Bypass
   MSet_Bypass15 : ALIAS FOR Wrk_MSet.15;   // Maint. Bypass Toggle for Interlock Cond. 15: 1=Bypass
   PCmd_Reset : BOOL;   // Program Command to Reset Latched Interlocks
   OCmd_Reset : BOOL;   // Operator Command to Reset Latched Interlocks
END_VAR
VAR_OUTPUT
   Sts_IntlkOK : BOOL := 1; {access Read Only, visible}   // Overall Interlock Status (1=OK to run, 0=Stop)
   Sts_NBIntlkOK : BOOL := 1; {access Read Only, visible}   // Non-Bypassable Interlock Status (1=All NB Interlocks OK to run)
   Sts_BypActive : BOOL; {access Read Only}   // 1=Interlock Bypassing is Active (ignore bypassable interlocks)
   Sts_Intlk : INT; {access Read Only, visible}   // Individual Interlock Status (1=Stop, 0=OK)
   Sts_FirstOut : INT; {access Read Only, visible}   // Interlock First Out Status (bit 1 is First Not-OK condition)
   Rdy_Reset : BOOL; {access Read Only}   // 1=Ready to receive OCmd_Reset (reset required)
   P_Intlk : BOOL;   // Unique Parameter Name for auto - discovery
END_VAR
VAR
   Cfg_CondTxt : STRING_20[16] := ([0] := 'Enter Description #0');   // Short HMI description of Interlock Conditions
   Wrk_Inp : INT;   // Collection copy of Inp_IntlkXXs
   Wrk_NB : INT; {access None}   // Working register for Non-Bypassable Interlock ogic
   Wrk_Intlk : INT; {access None}   // Working register for Interlock logic
   Wrk_FirstOut : INT; {access None}   // Working register for First Out logic
   Wrk_Sts : INT; {access None}   // Working register for generating Interlock status
   Wrk_PrevSts : INT; {access None}   // Interlock Status previous scan
   Wrk_LatchEnable : BOOL := 1; {access None}   // 1=Latch interlock if configured to latch, 0=don't latch
   Inf_Tab : SINT;   // Tab to display (FTView ME)
   Wrk_InpInv : INT; {access None}   // Input states after inversion based on Cfg_OKState
   Inf_Type : STRING_16 := 'P_Intlk'; {access Read Only}   // Type identifier for HMI navigation
   Cfg_Label : STRING_20 := 'Interlocks';   // Label for graphic symbol displayed on HMI
   Cfg_Tag : STRING_20 := 'P_Intlk';   // Tagname for display on HMI
   Cfg_Desc : STRING_40 := 'Interlocks with First Out';   // Description for display on HMI
   Cfg_NavTag : STRING_NavTag[16];   // Tagnames for destinations of Navigation buttons
   Inf_Lib : STRING_12 := 'RA-BAS'; {access Read Only}   // Display Library for Faceplate call-up
   Wrk_MSet : INT;   // Internal copy of individual condition Maint. Bypass toggles
   Wrk_NonIntlkStop : BOOL; {access None}   // One-Shot store: Stop OTHER than Interlock Stop occurred.
   Wrk_SetFirstOut : BOOL; {access None}   // One-Shot store: First Out update triggered
END_VAR

ROUTINE EnableInFalse   (* ladder *)
// Set summary "OK" Status bits to FALSE (0)
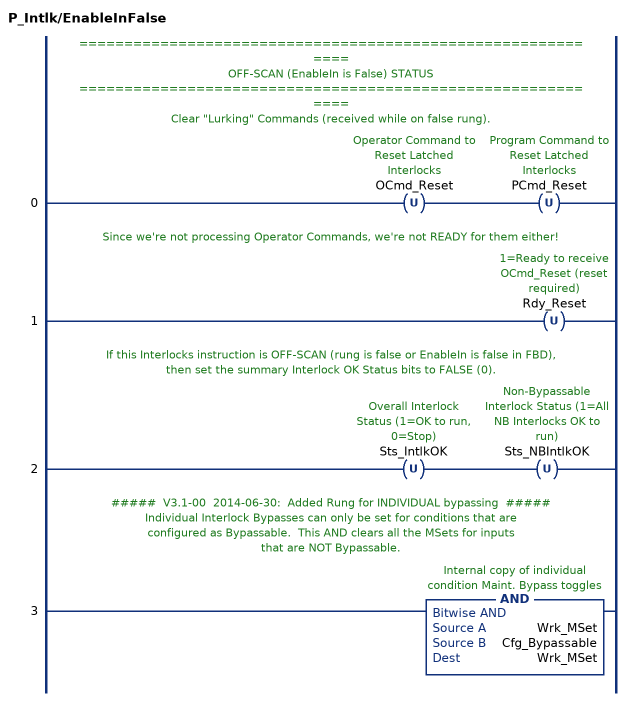
   // ============================================================
   // OFF-SCAN (EnableIn is False) STATUS
   // ============================================================
   //  Clear "Lurking" Commands (received while on false rung).
   0: OTU(OCmd_Reset)OTU(PCmd_Reset);
   // Since we're not processing Operator Commands, we're not READY for them either!
   1: OTU(Rdy_Reset);
   // If this Interlocks instruction is OFF-SCAN (rung is false or EnableIn is false in FBD),
   // then set the summary Interlock OK Status bits to FALSE (0).
   2: OTU(Sts_IntlkOK)OTU(Sts_NBIntlkOK);
   // #####  V3.1-00  2014-06-30:  Added Rung for INDIVIDUAL bypassing  #####
   // Individual Interlock Bypasses can only be set for conditions that are
   // configured as Bypassable.  This AND clears all the MSets for inputs
   // that are NOT Bypassable.
   3: AND(Wrk_MSet,Cfg_Bypassable,Wrk_MSet);
END_ROUTINE

ROUTINE Logic   (* ladder *)
// Check Interlock Conditions
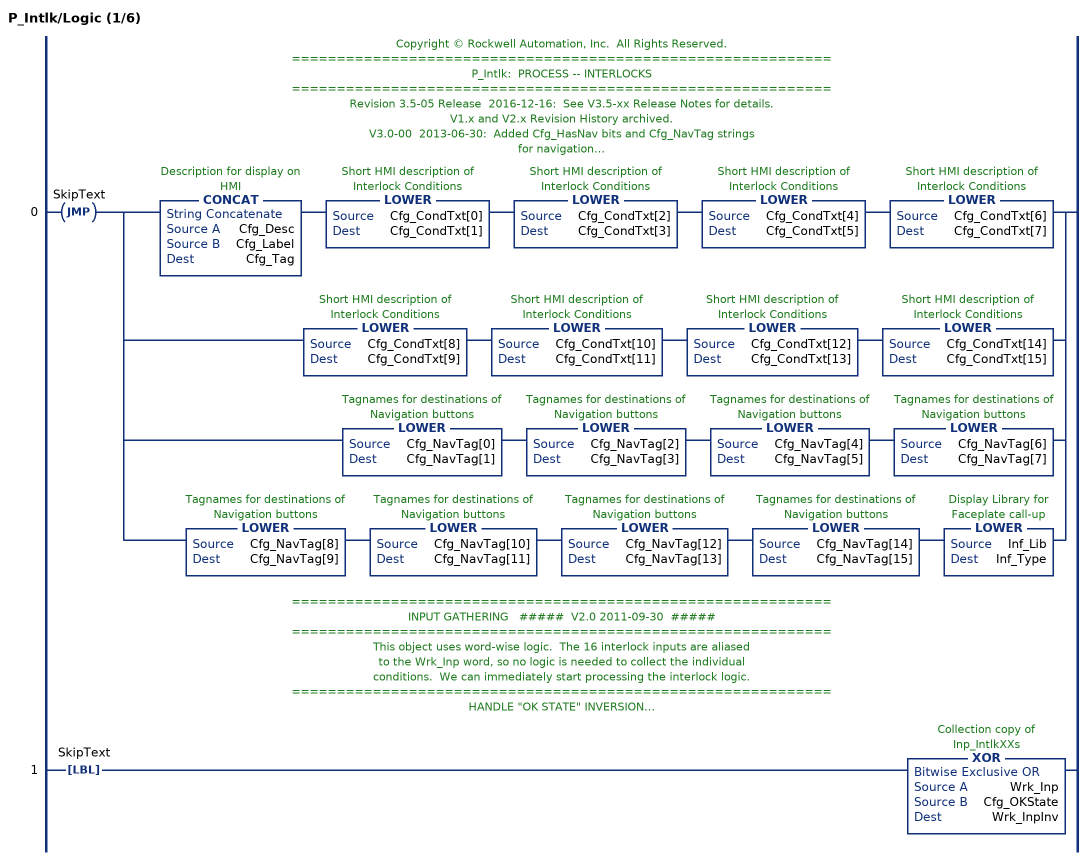
   // Copyright © Rockwell Automation, Inc.  All Rights Reserved.
   // ============================================================
   // P_Intlk:  PROCESS -- INTERLOCKS
   // ============================================================
   // Revision 3.5-05 Release  2016-12-16:  See V3.5-xx Release Notes for details.
   // V1.x and V2.x Revision History archived.
   // V3.0-00  2013-06-30:  Added Cfg_HasNav bits and Cfg_NavTag strings
   // for navigation.
   // V3.1-00  2014-06-30:  Modified to allow Maintenance to set up bypassing
   // of individual interlock conditions.
   // V3.1-01  2014-09-03:  Unmodified, up-rev only for V3.1-01 public release.
   // V3.5-01  2016-01-29:  Unmodified, up-rev only for V3.5.01 Release.
   // V3.5-05  2016-12-16:  Changed Nav Tags to user-defined STRING_NavTag type.
   // Modified logic to maintain First-Out indication until next stop.
   // ============================================================
   // This Instruction monitors up to 16 Interlock conditions.  It provides these features:
   // *  The "OK" state of each Interlock Input is configurable.
   // By default, each Input is 1 to trip, 0 when OK to run.
   // *  Interlocks may be configured as Latched.  Latched Interlocks
   // require a Reset Command to clear.  The latching function can be inhibited
   // via a Latch Defeat input, for example, to avoid latching Interlocks for a stopped motor.
   // *  Interlocks may be configured as Bypassable.  Bypassable Interlocks are reported
   // separately; the destination object can use this information to bypass these
   // Interlocks in Maintenance Mode or upon command.
   // *  First-Out reporting indicates the first condition that
   // caused the running equipment to be tripped.
   // * For each Interlock condition, a Tag may be defined for navigation. Clicking
   // the Interlock description will call up the associated Tag's Faceplate.
   // ============================================================
   // SHOW LOCAL STRINGS
   // ============================================================
   // The STRINGs containing the text associated with each instance of this
   // instruction cannot be Input or Output Parameters, because STRINGs are not
   //  'atomic' types. (Inputs and Outputs must be SINT, INT, DINT, REAL, or BOOL.)
   // In order to make it easier to find and configure these STRINGs, this rung
   // was added.  THE JMP (and the LBL on the following rung)
   // MUST NOT BE REMOVED!!!
   // To view the STRINGs, go to the instruction instance (in LD or FBD), RIGHT-click
   // to bring up the context menu and select "Open Instruction Logic".
   // This rung will appear with the STRING values for the selected instance.
   // You may double-click the STRING values here to modify them as well.
   // #####  V3.0-00  2013-06-30:  Added Cfg_NavTag strings on this rung  #####
   0: JMP(SkipText)[CONCAT(Cfg_Desc,Cfg_Label,Cfg_Tag) LOWER(Cfg_CondTxt[0],Cfg_CondTxt[1]) LOWER(Cfg_CondTxt[2],Cfg_CondTxt[3]) LOWER(Cfg_CondTxt[4],Cfg_CondTxt[5]) LOWER(Cfg_CondTxt[6],Cfg_CondTxt[7]) ,LOWER(Cfg_CondTxt[8],Cfg_CondTxt[9]) LOWER(Cfg_CondTxt[10],Cfg_CondTxt[11]) LOWER(Cfg_CondTxt[12],Cfg_CondTxt[13]) LOWER(Cfg_CondTxt[14],Cfg_CondTxt[15]) ,LOWER(Cfg_NavTag[0],Cfg_NavTag[1]) LOWER(Cfg_NavTag[2],Cfg_NavTag[3]) LOWER(Cfg_NavTag[4],Cfg_NavTag[5]) LOWER(Cfg_NavTag[6],Cfg_NavTag[7]) ,LOWER(Cfg_NavTag[8],Cfg_NavTag[9]) LOWER(Cfg_NavTag[10],Cfg_NavTag[11]) LOWER(Cfg_NavTag[12],Cfg_NavTag[13]) LOWER(Cfg_NavTag[14],Cfg_NavTag[15]) LOWER(Inf_Lib,Inf_Type) ];
   // ============================================================
   // INPUT GATHERING   #####  V2.0 2011-09-30  #####
   // ============================================================
   // This object uses word-wise logic.  The 16 interlock inputs are aliased
   // to the Wrk_Inp word, so no logic is needed to collect the individual
   // conditions.  We can immediately start processing the interlock logic.
   // ============================================================
   // HANDLE "OK STATE" INVERSIONS
   // ============================================================
   // This rung inverts the Input bits whose "OK State" is 1 (0 to Stop).
   // The resulting Wrk_Inp word is ZERO if all interlock inputs are "OK".
   1: LBL(SkipText)XOR(Wrk_Inp,Cfg_OKState,Wrk_InpInv);
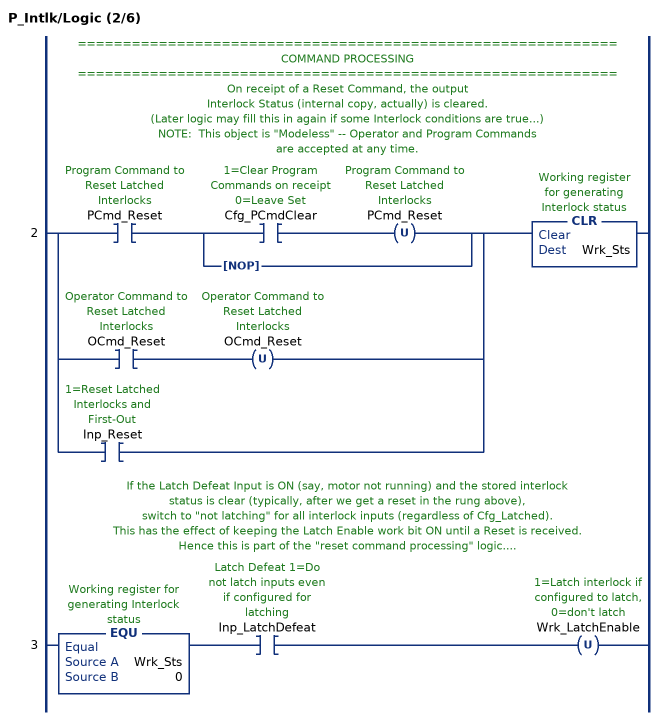
   // ============================================================
   // COMMAND PROCESSING
   // ============================================================
   // On receipt of a Reset Command, the output
   // Interlock Status (internal copy, actually) is cleared.
   // (Later logic may fill this in again if some Interlock conditions are true...)
   // NOTE:  This object is "Modeless" -- Operator and Program Commands
   // are accepted at any time.
   2: [XIC(PCmd_Reset) [XIC(Cfg_PCmdClear) OTU(PCmd_Reset) ,NOP() ] ,XIC(OCmd_Reset) OTU(OCmd_Reset) ,XIC(Inp_Reset) ]CLR(Wrk_Sts);
   // If the Latch Defeat Input is ON (say, motor not running) and the stored interlock
   // status is clear (typically, after we get a reset in the rung above),
   // switch to "not latching" for all interlock inputs (regardless of Cfg_Latched).
   // This has the effect of keeping the Latch Enable work bit ON until a Reset is received.
   // Hence this is part of the "reset command processing" logic....
   3: EQU(Wrk_Sts,0)XIC(Inp_LatchDefeat)OTU(Wrk_LatchEnable);
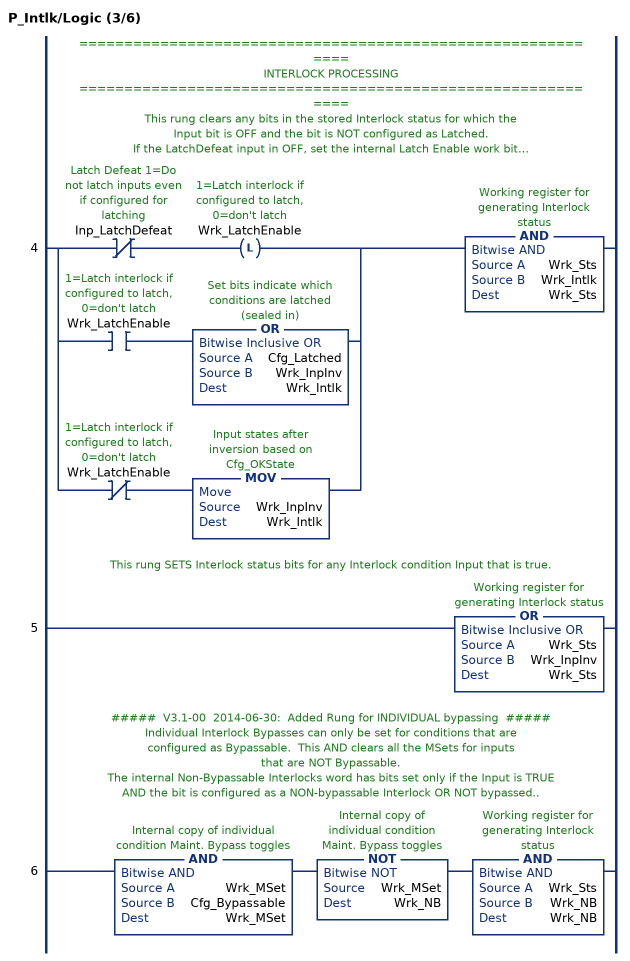
   // ============================================================
   // INTERLOCK PROCESSING
   // ============================================================
   // This rung clears any bits in the stored Interlock status for which the
   // Input bit is OFF and the bit is NOT configured as Latched.
   // If the LatchDefeat input in OFF, set the internal Latch Enable work bit.
   // If this bit is ON, don't clear any latched bits with this rung (keep them latched).
   // If this bit is OFF, clear any bits that are NOT on in the input, whether
   // configured for latching or not!
   4: [XIO(Inp_LatchDefeat) OTL(Wrk_LatchEnable) ,XIC(Wrk_LatchEnable) OR(Cfg_Latched,Wrk_InpInv,Wrk_Intlk) ,XIO(Wrk_LatchEnable) MOV(Wrk_InpInv,Wrk_Intlk) ]AND(Wrk_Sts,Wrk_Intlk,Wrk_Sts);
   // This rung SETS Interlock status bits for any Interlock condition Input that is true.
   5: OR(Wrk_Sts,Wrk_InpInv,Wrk_Sts);
   // #####  V3.1-00  2014-06-30:  Added Rung for INDIVIDUAL bypassing  #####
   // Individual Interlock Bypasses can only be set for conditions that are
   // configured as Bypassable.  This AND clears all the MSets for inputs
   // that are NOT Bypassable.
   // The internal Non-Bypassable Interlocks word has bits set only if the Input is TRUE
   // AND the bit is configured as a NON-bypassable Interlock OR NOT bypassed..
   6: AND(Wrk_MSet,Cfg_Bypassable,Wrk_MSet)NOT(Wrk_MSet,Wrk_NB)AND(Wrk_Sts,Wrk_NB,Wrk_NB);
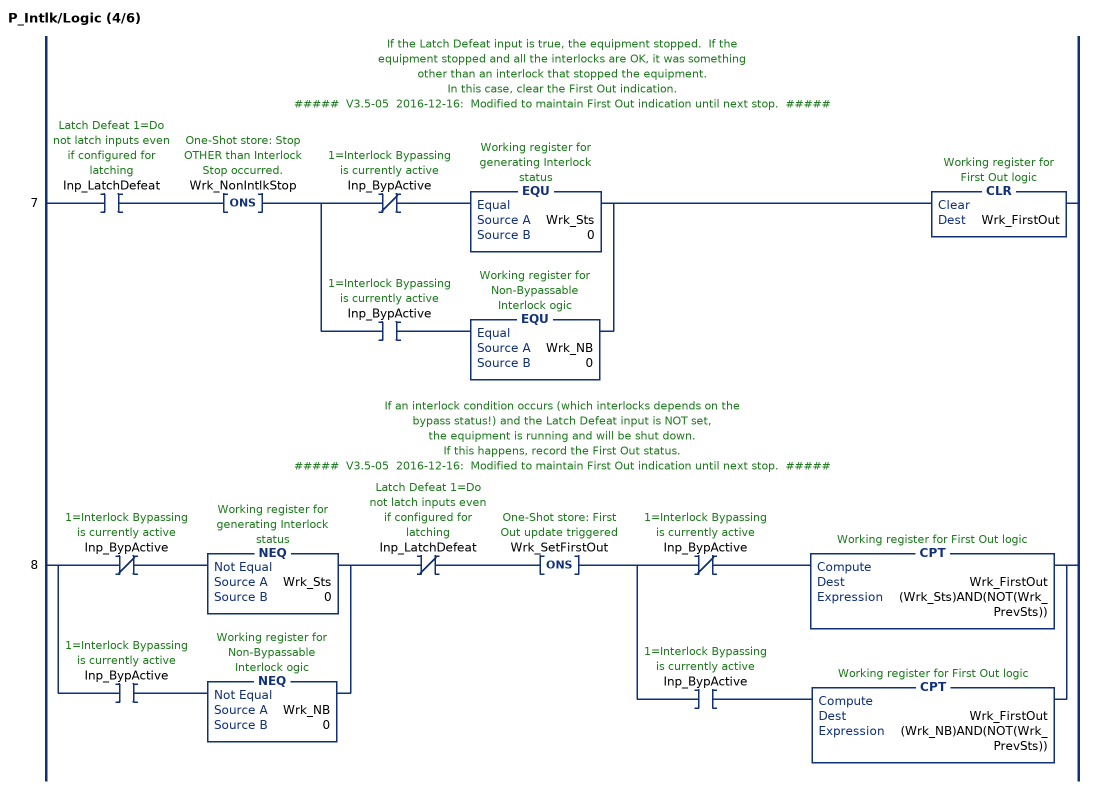
   // If the Latch Defeat input is true, the equipment stopped.  If the
   // equipment stopped and all the interlocks are OK, it was something
   // other than an interlock that stopped the equipment.
   // In this case, clear the First Out indication.
   // #####  V3.5-05  2016-12-16:  Modified to maintain First Out indication until next stop.  #####
   7: XIC(Inp_LatchDefeat)ONS(Wrk_NonIntlkStop)[XIO(Inp_BypActive) EQU(Wrk_Sts,0) ,XIC(Inp_BypActive) EQU(Wrk_NB,0) ]CLR(Wrk_FirstOut);
   // If an interlock condition occurs (which interlocks depends on the
   // bypass status!) and the Latch Defeat input is NOT set,
   // the equipment is running and will be shut down.
   // If this happens, record the First Out status.
   // #####  V3.5-05  2016-12-16:  Modified to maintain First Out indication until next stop.  #####
   8: [XIO(Inp_BypActive) NEQ(Wrk_Sts,0) ,XIC(Inp_BypActive) NEQ(Wrk_NB,0) ]XIO(Inp_LatchDefeat)ONS(Wrk_SetFirstOut)[XIO(Inp_BypActive) CPT(Wrk_FirstOut,(Wrk_Sts)AND(NOT(Wrk_PrevSts))) ,XIC(Inp_BypActive) CPT(Wrk_FirstOut,(Wrk_NB)AND(NOT(Wrk_PrevSts))) ];
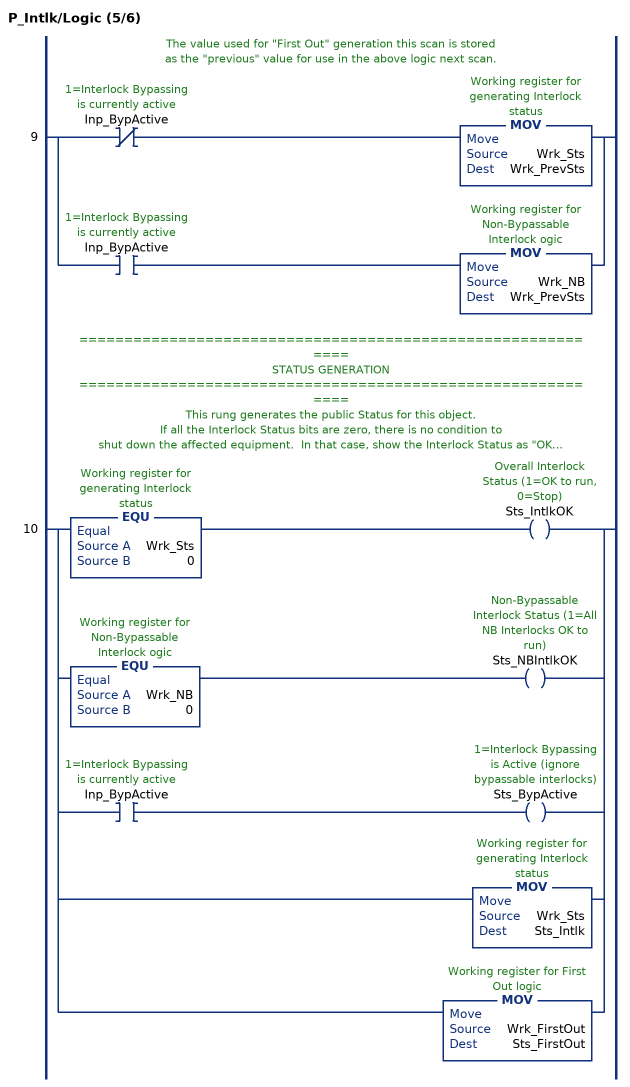
   // The value used for "First Out" generation this scan is stored
   // as the "previous" value for use in the above logic next scan.
   9: [XIO(Inp_BypActive) MOV(Wrk_Sts,Wrk_PrevSts) ,XIC(Inp_BypActive) MOV(Wrk_NB,Wrk_PrevSts) ];
   // ============================================================
   // STATUS GENERATION
   // ============================================================
   // This rung generates the public Status for this object.
   // If all the Interlock Status bits are zero, there is no condition to
   // shut down the affected equipment.  In that case, show the Interlock Status as "OK"
   // Similar logic applies for the Non-Bypassable Interlocks OK Status.
   // Also show the individual Interlock Status bits and the First Out Status bits.
   // NOTE:  Working registers are used to prevent outside writes to the Sts_xxx
   // parameters from affecting the state of this object!
   10: [[EQU(Wrk_Sts,0) OTE(Sts_IntlkOK) ,EQU(Wrk_NB,0) OTE(Sts_NBIntlkOK) ] ,XIC(Inp_BypActive) OTE(Sts_BypActive) ,MOV(Wrk_Sts,Sts_Intlk) ,MOV(Wrk_FirstOut,Sts_FirstOut) ];
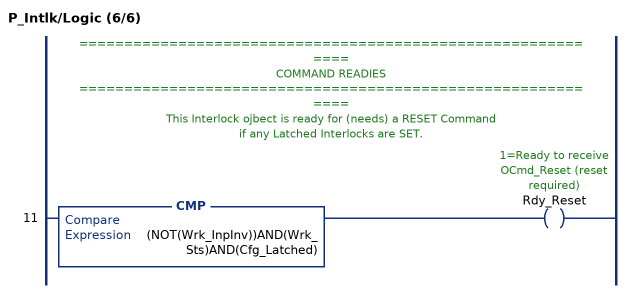
   // ============================================================
   // COMMAND READIES
   // ============================================================
   // This Interlock ojbect is ready for (needs) a RESET Command
   // if any Latched Interlocks are SET.
   11: CMP((NOT(Wrk_InpInv))AND(Wrk_Sts)AND(Cfg_Latched))OTE(Rdy_Reset);
END_ROUTINE
